{attribute addProperty BoxType "EPP1816-3008-0016"}
{attribute addProperty Id "InputAT %I*ARRAY[0 ..7] OF BOOL6480"}
{attribute addProperty CRC "1701588874"}
{attribute addProperty SizeInBites "64"}
{attribute addProperty SizeInBytes "8"}
TYPE DIG_Inputs_Channel_628B507D :
STRUCT
	{attribute addProperty Name "Input"}
	Input AT %I* : ARRAY[0 ..7] OF BOOL;
END_STRUCT
END_TYPE

(* stored: Version 1.2.0.0, ProductVersion 3.1.4024.9
   DUT DIG_Inputs_Channel_628B507D: Id {2771f78c-9461-4cbe-9f36-463685537141} *)
